FUNCTION_BLOCK A2X_AND_2 (* Composite FB to calculate boolean AND between 2 A2X adapters (UP and DOWN independently) *)
  (* Standard: 61499-2; Function: OUT.UP = IN1.UP AND IN2.UP, OUT.DOWN = IN1.DOWN AND IN2.DOWN; Description: Copyright (c) 2026 HR Agrartechnik GmbH This program and the accompanying materials are made available under the terms of the Eclipse Public License 2.0 which is available at https://www.eclipse.org/legal/epl-2.0/ SPDX-License-Identifier: EPL-2.0 *)
  (* Version 1.0, 2026-08-31, Franz Höpfinger, HR Agrartechnik GmbH, Initial Version *)
  PACKAGE adapter::booleanOperators;
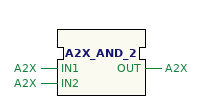
  SOCKETS
    IN1 : adapter::types::unidirectional::A2X; (* AND input 1 *)
    IN2 : adapter::types::unidirectional::A2X; (* AND input 2 *)
  END_SOCKETS
  PLUGS
    OUT : adapter::types::unidirectional::A2X; (* AND result *)
  END_PLUGS
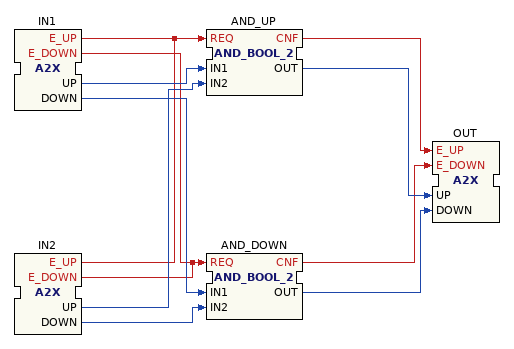
  FBS
    AND_UP : iec61131::booleanOperators::AND_BOOL_2; (* ANDs the UP channel *)
    AND_DOWN : iec61131::booleanOperators::AND_BOOL_2; (* ANDs the DOWN channel *)
  END_FBS
  EVENT_CONNECTIONS
    IN1.E_UP TO AND_UP.REQ;
    IN2.E_UP TO AND_UP.REQ;
    AND_UP.CNF TO OUT.E_UP;
    IN1.E_DOWN TO AND_DOWN.REQ;
    IN2.E_DOWN TO AND_DOWN.REQ;
    AND_DOWN.CNF TO OUT.E_DOWN;
  END_CONNECTIONS
  DATA_CONNECTIONS
    IN1.UP TO AND_UP.IN1;
    IN2.UP TO AND_UP.IN2;
    AND_UP.OUT TO OUT.UP;
    IN1.DOWN TO AND_DOWN.IN1;
    IN2.DOWN TO AND_DOWN.IN2;
    AND_DOWN.OUT TO OUT.DOWN;
  END_CONNECTIONS
END_FUNCTION_BLOCK
